FUNCTION_BLOCK StopMovementsAndProgramTask EXTENDS TcoCore.TcoTask 
VAR

	_stopType: TcoAbstractions.eTcoRoboticsStopType;
END_VAR
VAR
    {attribute 'hide'} 
	_progress : INT := 0;
    {attribute 'hide'} 
	_infoTimer :  TON;
    {attribute 'hide'} 
	_errorTimer :  TON;
    {attribute 'hide'} 
	_varInfo : __SYSTEM.VAR_INFO;
    {attribute 'hide'} 
	_sb : TcoCore.StringBuilder;
END_VAR

VAR_IN_OUT
    inoConfig 	: TcoIrc5_Config_v_1_x_x;
	inoControl 	: TcoIrc5_Control_v_1_x_x;
	inoStatus 	: TcoIrc5_Status_v_1_x_x;	
END_VAR



IF Execute() THEN
	IF _progress = 0 THEN
		IF NOT __ISVALIDREF(inoControl) THEN
			_varInfo :=__VARINFO(inoControl);
			Messenger.Programming(_sb.Clear().Append('<#Invalid reference: #>').Append(_varInfo.Symbol).ToString()).Pin();
		ELSIF NOT __ISVALIDREF(inoConfig) THEN                                                  
			_varInfo :=__VARINFO(inoConfig);                                                    
			Messenger.Programming(_sb.Clear().Append('<#Invalid reference: #>').Append(_varInfo.Symbol).ToString()).Pin();
		ELSIF NOT __ISVALIDREF(inoStatus) THEN                                                  
			_varInfo :=__VARINFO(inoStatus);                                                    
			Messenger.Programming(_sb.Clear().Append('<#Invalid reference: #>').Append(_varInfo.Symbol).ToString()).Pin();
			ELSE
			_progress := _progress + 1;
		END_IF

	END_IF
	IF _progress = 1 THEN
		inoControl.SoftStop := TRUE;
		inoControl.QuickStop := FALSE;
	
		IF _stopType = TcoAbstractions.eTcoRoboticsStopType.Quick THEN
			inoControl.SoftStop := TRUE;
			inoControl.QuickStop := FALSE;
		END_IF
		IF inoStatus.State.MoveInactive THEN
			_progress := _progress + 1;
		END_IF
	END_IF;		

	IF _progress = 2 THEN
		inoControl.StopProgram:=TRUE;
		IF NOT inoStatus.State.CycleOn THEN
			_progress := _progress + 1;
		END_IF
	END_IF;		
	
	IF _progress = 3 THEN	
		inoControl.SoftStop := FALSE;
		inoControl.QuickStop := FALSE;
		inoControl.StopProgram:=FALSE;
	END_IF;		
		

    DoneWhen(_progress=3 AND  inoStatus.State.MoveInactive AND NOT inoStatus.State.CycleOn);
    CallTimers(TRUE);
	
	THIS^.ThrowWhen(_errorTimer.Q);
END_IF

METHOD CallTimers
VAR_INPUT
	inValue : BOOL;
END_VAR
IF  __ISVALIDREF(inoConfig) THEN  
_infoTimer(IN := inValue, PT := THIS^.inoConfig.InfoTime);
_errorTimer(IN := inValue, PT := THIS^.inoConfig.ErrorTime);
END_IF;
END_METHOD

METHOD PUBLIC FB_init : BOOL
VAR_INPUT
    bInitRetains : BOOL; // if TRUE, the retain variables are initialized (warm start / cold start)
    bInCopyCode : BOOL; // if TRUE, the instance afterwards gets moved into the copy code (online change)
  	ParentObject : ITcoObject;	
END_VAR
END_METHOD

METHOD INTERNAL InvokeWithParams : ITcoTaskStatus
VAR_INPUT
	inStopType : eTcoRoboticsStopType;
END_VAR
_stopType := inStopType;
InvokeWithParams := THIS^.Invoke();
END_METHOD

(*~
	<docu>
		<summary>
			Executes when task is aborted.
		</summary>			
	</docu>	
~*)
METHOD PROTECTED OnAbort
IF  __ISVALIDREF(inoStatus) THEN   THIS^.inoStatus.ActionDescription := '<#Stop movements and program was aborted, while not yet completed!#>';END_IF;
END_METHOD

(*~
	<docu>
		<summary>
			Executes when task reaches the ```Done``` state .
		</summary>			
	</docu>	
~*)
METHOD PROTECTED OnDone
IF  __ISVALIDREF(inoStatus) THEN  THIS^.inoStatus.ActionDescription := '<#Stop movements and program  was completed successfully.#>';END_IF;
END_METHOD

(*~
	<docu>
		<summary>
			Executes when task reaches the ```Error``` state.
			<para>
				Do not confuse with <see cref="PlcDocu.TcoCore.TcoTask.WhileError()"/>, that is called cyclically until '''Error''' state is left.
			</para>
		</summary>			
	</docu>	
~*)
METHOD PROTECTED OnError
IF  __ISVALIDREF(inoStatus) THEN   THIS^.inoStatus.ActionDescription := '<#Stop movements and program finished with error.#>'; END_IF;
END_METHOD

METHOD PROTECTED OnStart
IF  __ISVALIDREF(inoStatus) THEN  THIS^.inoStatus.ActionDescription := '<#Stop movements and program started.#>'; END_IF;
END_METHOD

(*~
	<docu>
		<summary>
			Restores this instance to the Ready state. Can be called explicitly or from within one of the restore mechanisms.
			<para>
				See also <see cref="PlcDocu.TcoCore.TcoTask.AutoRestorable()"/>
			</para>
		</summary>			
	</docu>	
~*)
METHOD Restore : ITcoRestorable
SUPER^.Restore();
_progress := 0;
CallTimers(FALSE);
Messenger.UnPin();
END_METHOD

END_FUNCTION_BLOCK

(* stored: Version 1.1.0.1, ProductVersion 3.1.4024.12
   POU StopMovementsAndProgramTask: Id {bbc19dcc-9bcd-0b3f-09de-7073c12da196}, SpecialFunc None
   Method CallTimers: Id {c2c8e197-caad-09a4-0d01-3ffe9e49e499}
   Method FB_init: Id {fe08e306-c22d-0e6b-3c13-63ab1d6fa1bb}
   Method InvokeWithParams: Id {94750881-5ca5-0421-012f-835b9aa7a2b0}
   Method OnAbort: Id {6e6849be-c1e2-0cb8-00f0-d18e388fb8f8}
   Method OnDone: Id {51a8987e-1e66-08ef-1570-d67484cf25a2}
   Method OnError: Id {22f3ae59-de11-0e7f-2631-bb6d0b4b63fd}
   Method OnStart: Id {23130bcb-8225-07f0-048a-2722a360db86}
   Method Restore: Id {f6e004b9-78ef-0f57-24a2-3a86a8d50611} *)
